// TIA Portal project "EJERCICIOS CON LAS ES ANALÓGICAS" (V15.1)

(* hardware
DEVICE "S7-1200 station_1"  S7-1200 Station
   slot 0: "Rack_0"  S7-1200 Rack  Rack  V1.0
   slot 1: "PLC_1"  CPU 1214C AC/DC/Rly  6ES7 214-1BG40-0XB0  V4.1
*)

// ===== PLC "PLC_1"  CPU 1214C AC/DC/Rly =====

VAR_GLOBAL   // PLC tag table "Tabla de variables estándar"
   "Tag_1" AT %IW64 : Int;
   "Tag_2" AT %MD40 : Real;
   "Tag_3" AT %MD44 : Real;
   "Tag_4" AT %MD80 : Real;
   "Tag_5" AT %MD81 : Real;
   "Tag_6" AT %IW67 : Int;
   "Tag_7" AT %IW66 : Int;
   "Tag_8" AT %MD84 : Real;
   "Tag_9" AT %M500.0 : Bool;
END_VAR

ORGANIZATION_BLOCK "Main"   // OB1, LAD, ProgramCycle
TITLE = "Main Program Sweep (Cycle)"
{ S7_Optimized_Access := 'TRUE' }
VERSION : 0.1
BEGIN

REGION Network 1
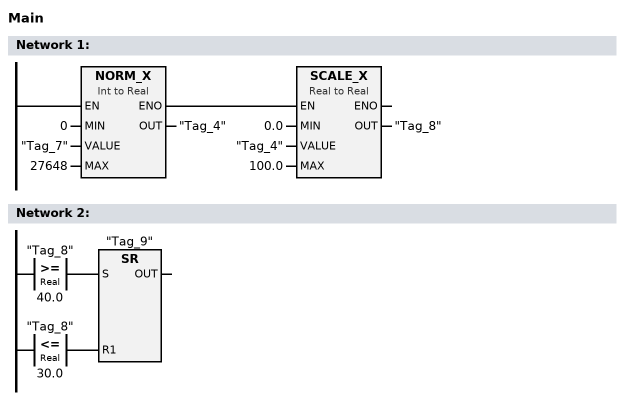
   RUNG wire#powerrail
      { S7_Templates := "[SrcType := Int, DestType := Real]"; S7_GenerateENO := "TRUE" } Normalize(min := 0, value := "Tag_7", max := 27648, out => "Tag_4")
      { S7_Templates := "[SrcType := Real, DestType := Real]"; S7_GenerateENO := "TRUE" } Scale(min := 0.0, value := "Tag_4", max := 100.0, out => "Tag_8")
   END_RUNG
   // the same network as SCL:
   // ENO of a box is taken as its EN; it also drops when the box reports an error
   "Tag_4" := NORM_X(MIN := 0, VALUE := "Tag_7", MAX := 27648);
   "Tag_8" := SCALE_X(MIN := 0.0, VALUE := "Tag_4", MAX := 100.0);
END_REGION

REGION Network 2
   RUNG wire#powerrail
      { S7_Templates := "SrcType := Real" } GE_Contact(in1 := "Tag_8", in2 := 40.0)
      S_SR(operand := "Tag_9", r1 := wire#w1)
   END_RUNG
   RUNG wire#powerrail
      { S7_Templates := "SrcType := Real" } LE_Contact(in1 := "Tag_8", in2 := 30.0)
   END_RUNG wire#w1
   // the same network as SCL:
   IF "Tag_8" >= 40.0 THEN
       "Tag_9" := TRUE;   // SR flip-flop
   END_IF;
   IF "Tag_8" <= 30.0 THEN "Tag_9" := FALSE; END_IF;
END_REGION
END_ORGANIZATION_BLOCK